FUNCTION_BLOCK Positions_init
VAR_INPUT
END_VAR
VAR_OUTPUT
END_VAR
VAR
	Current_Position: Array [0..10] of Places_position;
END_VAR

Current_Position[0].Number:=0;
Current_Position[0].Coordinate_X_Axis:=Positions.Position_1;
Current_Position[0].Coordinate_Y_Axis:=Positions.Position_2;

Current_Position[1].Number:=0;
Current_Position[1].Coordinate_X_Axis:=Positions.Position_1;
Current_Position[1].Coordinate_Y_Axis:=Positions.Position_2;

Current_Position[2].Number:=0;
Current_Position[2].Coordinate_X_Axis:=Positions.Position_1;
Current_Position[2].Coordinate_Y_Axis:=Positions.Position_2;

Current_Position[3].Number:=0;
Current_Position[3].Coordinate_X_Axis:=Positions.Position_1;
Current_Position[3].Coordinate_Y_Axis:=Positions.Position_2;

Current_Position[4].Number:=0;
Current_Position[4].Coordinate_X_Axis:=Positions.Position_1;
Current_Position[4].Coordinate_Y_Axis:=Positions.Position_2;

Current_Position[5].Number:=0;
Current_Position[5].Coordinate_X_Axis:=Positions.Position_1;
Current_Position[5].Coordinate_Y_Axis:=Positions.Position_2;

Current_Position[6].Number:=0;
Current_Position[6].Coordinate_X_Axis:=Positions.Position_1;
Current_Position[6].Coordinate_Y_Axis:=Positions.Position_2;

Current_Position[7].Number:=0;
Current_Position[7].Coordinate_X_Axis:=Positions.Position_1;
Current_Position[7].Coordinate_Y_Axis:=Positions.Position_2;

Current_Position[8].Number:=0;
Current_Position[8].Coordinate_X_Axis:=Positions.Position_1;
Current_Position[8].Coordinate_Y_Axis:=Positions.Position_2;

Current_Position[9].Number:=0;
Current_Position[9].Coordinate_X_Axis:=Positions.Position_1;
Current_Position[9].Coordinate_Y_Axis:=Positions.Position_2;

Current_Position[10].Number:=0;
Current_Position[10].Coordinate_X_Axis:=Positions.Position_1;
Current_Position[10].Coordinate_Y_Axis:=Positions.Position_2;

END_FUNCTION_BLOCK

(* stored: Version 1.1.0.1, ProductVersion 3.1.4024.11
   POU Positions_init: Id {d40c313c-a4a0-4c19-a065-c5edb0e93e52}, SpecialFunc None *)
